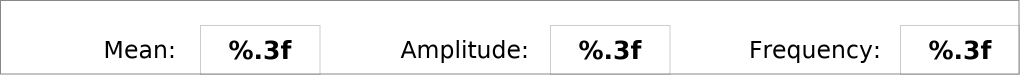
VISUALIZATION VISU_Sine  // 1020x75
    Textfield (200,25 120x50), "%.3f"
        OnMouseClick: write the text variable via InputWithLimits, min 0.1, max 0.7
    Textfield (80,25 120x50), "Mean:"
    Textfield (550,25 120x50), "%.3f"
        OnMouseClick: write the text variable via InputWithLimits, max 0.2
    Textfield (390,25 150x50), "Amplitude:"
    Textfield (900,25 120x50), "%.3f"
        OnMouseClick: write the text variable via Edit
    Textfield (740,25 150x50), "Frequency:"
END_VISUALIZATION
